NETWORK
TITLE = CALL SFC UO_MX_CIP if CIP running
//------------------------------------------------------------------------//
// SFC CALL   SFC CALL   SFC CALL   SFC CALL   SFC CALL   SFC CALL   SFC  //
//                                                                        //
// Call the SFC function if this is the running substate. This has to be  //
// called even if the block is not running so the SFC can process all     //
// commmands:                                                             //
//------------------------------------------------------------------------//
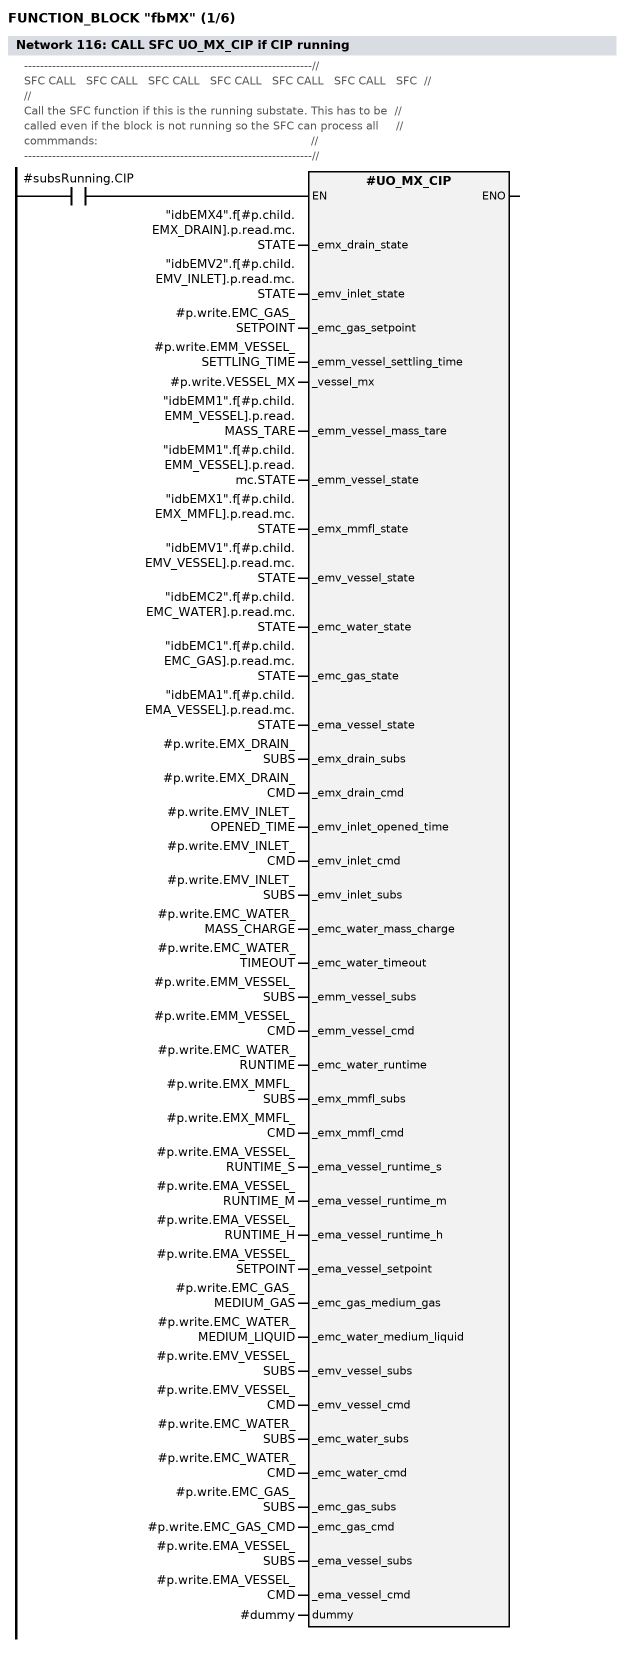
      A #subsRunning.CIP;
      JCN _notSFC_1_CIP;
      CALL #UO_MX_CIP
      (  _emx_drain_state            := "idbEMX4".f[#p.child.EMX_DRAIN].p.read.mc.STATE ,
         _emv_inlet_state            := "idbEMV2".f[#p.child.EMV_INLET].p.read.mc.STATE ,
         _emc_gas_setpoint           := #p.write.EMC_GAS_SETPOINT ,
         _emm_vessel_settling_time   := #p.write.EMM_VESSEL_SETTLING_TIME ,
         _vessel_mx                  := #p.write.VESSEL_MX ,
         _emm_vessel_mass_tare       := "idbEMM1".f[#p.child.EMM_VESSEL].p.read.MASS_TARE ,
         _emm_vessel_state           := "idbEMM1".f[#p.child.EMM_VESSEL].p.read.mc.STATE ,
         _emx_mmfl_state             := "idbEMX1".f[#p.child.EMX_MMFL].p.read.mc.STATE ,
         _emv_vessel_state           := "idbEMV1".f[#p.child.EMV_VESSEL].p.read.mc.STATE ,
         _emc_water_state            := "idbEMC2".f[#p.child.EMC_WATER].p.read.mc.STATE ,
         _emc_gas_state              := "idbEMC1".f[#p.child.EMC_GAS].p.read.mc.STATE ,
         _ema_vessel_state           := "idbEMA1".f[#p.child.EMA_VESSEL].p.read.mc.STATE ,
         _emx_drain_subs             := #p.write.EMX_DRAIN_SUBS ,
         _emx_drain_cmd              := #p.write.EMX_DRAIN_CMD ,
         _emv_inlet_opened_time      := #p.write.EMV_INLET_OPENED_TIME ,
         _emv_inlet_cmd              := #p.write.EMV_INLET_CMD ,
         _emv_inlet_subs             := #p.write.EMV_INLET_SUBS ,
         _emc_water_mass_charge      := #p.write.EMC_WATER_MASS_CHARGE ,
         _emc_water_timeout          := #p.write.EMC_WATER_TIMEOUT ,
         _emm_vessel_subs            := #p.write.EMM_VESSEL_SUBS ,
         _emm_vessel_cmd             := #p.write.EMM_VESSEL_CMD ,
         _emc_water_runtime          := #p.write.EMC_WATER_RUNTIME ,
         _emx_mmfl_subs              := #p.write.EMX_MMFL_SUBS ,
         _emx_mmfl_cmd               := #p.write.EMX_MMFL_CMD ,
         _ema_vessel_runtime_s       := #p.write.EMA_VESSEL_RUNTIME_S ,
         _ema_vessel_runtime_m       := #p.write.EMA_VESSEL_RUNTIME_M ,
         _ema_vessel_runtime_h       := #p.write.EMA_VESSEL_RUNTIME_H ,
         _ema_vessel_setpoint        := #p.write.EMA_VESSEL_SETPOINT ,
         _emc_gas_medium_gas         := #p.write.EMC_GAS_MEDIUM_GAS ,
         _emc_water_medium_liquid    := #p.write.EMC_WATER_MEDIUM_LIQUID ,
         _emv_vessel_subs            := #p.write.EMV_VESSEL_SUBS ,
         _emv_vessel_cmd             := #p.write.EMV_VESSEL_CMD ,
         _emc_water_subs             := #p.write.EMC_WATER_SUBS ,
         _emc_water_cmd              := #p.write.EMC_WATER_CMD ,
         _emc_gas_subs               := #p.write.EMC_GAS_SUBS ,
         _emc_gas_cmd                := #p.write.EMC_GAS_CMD ,
         _ema_vessel_subs            := #p.write.EMA_VESSEL_SUBS ,
         _ema_vessel_cmd             := #p.write.EMA_VESSEL_CMD ,
         dummy                       := #dummy
      );
_notSFC_1_CIP:      NOP 0;
NETWORK
TITLE = CALL SFC UO_MX_FILL if FILL running
//------------------------------------------------------------------------//
// SFC CALL   SFC CALL   SFC CALL   SFC CALL   SFC CALL   SFC CALL   SFC  //
//                                                                        //
// Call the SFC function if this is the running substate. This has to be  //
// called even if the block is not running so the SFC can process all     //
// commmands:                                                             //
//------------------------------------------------------------------------//
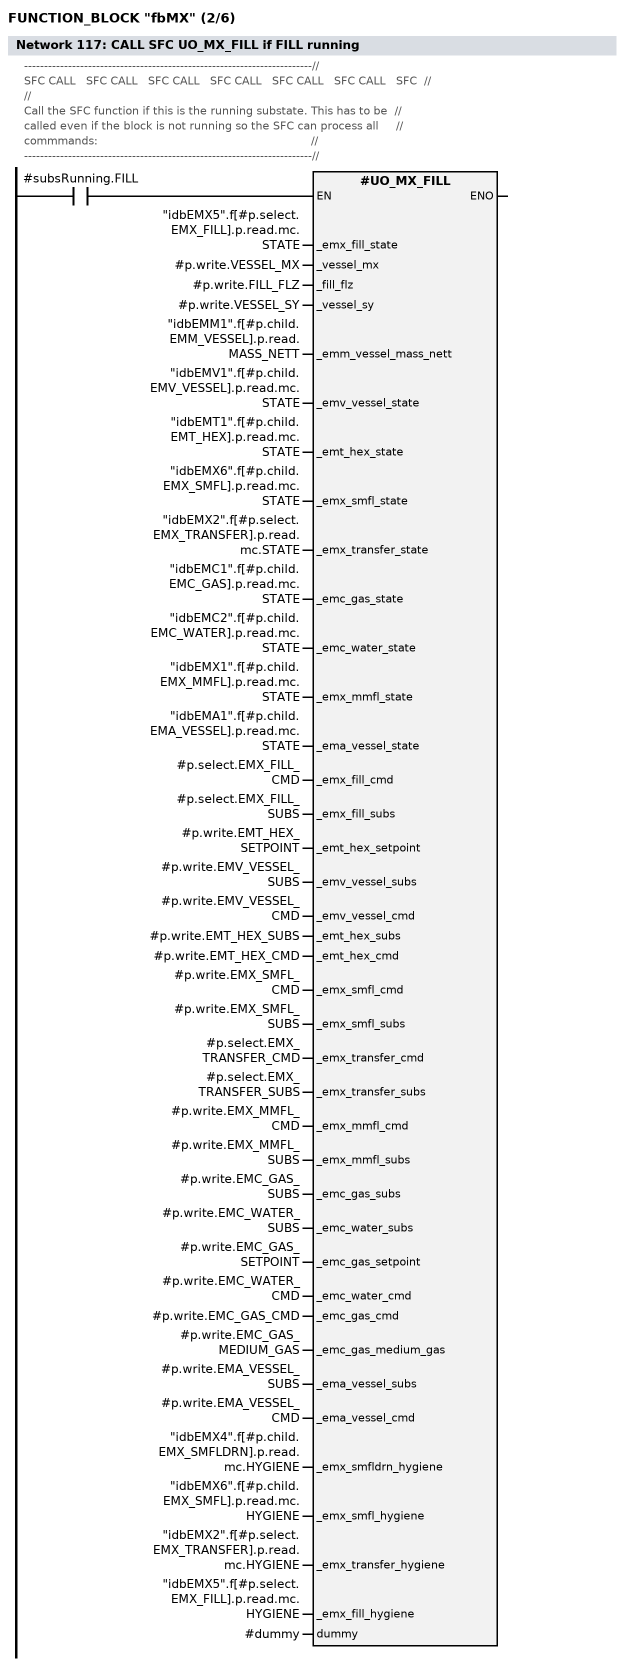
      A #subsRunning.FILL;
      JCN _notSFC_5_FILL;
      CALL #UO_MX_FILL
      (  _emx_fill_state             := "idbEMX5".f[#p.select.EMX_FILL].p.read.mc.STATE ,
         _vessel_mx                  := #p.write.VESSEL_MX ,
         _fill_flz                   := #p.write.FILL_FLZ ,
         _vessel_sy                  := #p.write.VESSEL_SY ,
         _emm_vessel_mass_nett       := "idbEMM1".f[#p.child.EMM_VESSEL].p.read.MASS_NETT ,
         _emv_vessel_state           := "idbEMV1".f[#p.child.EMV_VESSEL].p.read.mc.STATE ,
         _emt_hex_state              := "idbEMT1".f[#p.child.EMT_HEX].p.read.mc.STATE ,
         _emx_smfl_state             := "idbEMX6".f[#p.child.EMX_SMFL].p.read.mc.STATE ,
         _emx_transfer_state         := "idbEMX2".f[#p.select.EMX_TRANSFER].p.read.mc.STATE ,
         _emc_gas_state              := "idbEMC1".f[#p.child.EMC_GAS].p.read.mc.STATE ,
         _emc_water_state            := "idbEMC2".f[#p.child.EMC_WATER].p.read.mc.STATE ,
         _emx_mmfl_state             := "idbEMX1".f[#p.child.EMX_MMFL].p.read.mc.STATE ,
         _ema_vessel_state           := "idbEMA1".f[#p.child.EMA_VESSEL].p.read.mc.STATE ,
         _emx_fill_cmd               := #p.select.EMX_FILL_CMD ,
         _emx_fill_subs              := #p.select.EMX_FILL_SUBS ,
         _emt_hex_setpoint           := #p.write.EMT_HEX_SETPOINT ,
         _emv_vessel_subs            := #p.write.EMV_VESSEL_SUBS ,
         _emv_vessel_cmd             := #p.write.EMV_VESSEL_CMD ,
         _emt_hex_subs               := #p.write.EMT_HEX_SUBS ,
         _emt_hex_cmd                := #p.write.EMT_HEX_CMD ,
         _emx_smfl_cmd               := #p.write.EMX_SMFL_CMD ,
         _emx_smfl_subs              := #p.write.EMX_SMFL_SUBS ,
         _emx_transfer_cmd           := #p.select.EMX_TRANSFER_CMD ,
         _emx_transfer_subs          := #p.select.EMX_TRANSFER_SUBS ,
         _emx_mmfl_cmd               := #p.write.EMX_MMFL_CMD ,
         _emx_mmfl_subs              := #p.write.EMX_MMFL_SUBS ,
         _emc_gas_subs               := #p.write.EMC_GAS_SUBS ,
         _emc_water_subs             := #p.write.EMC_WATER_SUBS ,
         _emc_gas_setpoint           := #p.write.EMC_GAS_SETPOINT ,
         _emc_water_cmd              := #p.write.EMC_WATER_CMD ,
         _emc_gas_cmd                := #p.write.EMC_GAS_CMD ,
         _emc_gas_medium_gas         := #p.write.EMC_GAS_MEDIUM_GAS ,
         _ema_vessel_subs            := #p.write.EMA_VESSEL_SUBS ,
         _ema_vessel_cmd             := #p.write.EMA_VESSEL_CMD ,
         _emx_smfldrn_hygiene        := "idbEMX4".f[#p.child.EMX_SMFLDRN].p.read.mc.HYGIENE ,
         _emx_smfl_hygiene           := "idbEMX6".f[#p.child.EMX_SMFL].p.read.mc.HYGIENE ,
         _emx_transfer_hygiene       := "idbEMX2".f[#p.select.EMX_TRANSFER].p.read.mc.HYGIENE ,
         _emx_fill_hygiene           := "idbEMX5".f[#p.select.EMX_FILL].p.read.mc.HYGIENE ,
         dummy                       := #dummy
      );
_notSFC_5_FILL:      NOP 0;
NETWORK
TITLE = CALL SFC UO_MX_FILTER if FILTER running
//------------------------------------------------------------------------//
// SFC CALL   SFC CALL   SFC CALL   SFC CALL   SFC CALL   SFC CALL   SFC  //
//                                                                        //
// Call the SFC function if this is the running substate. This has to be  //
// called even if the block is not running so the SFC can process all     //
// commmands:                                                             //
//------------------------------------------------------------------------//
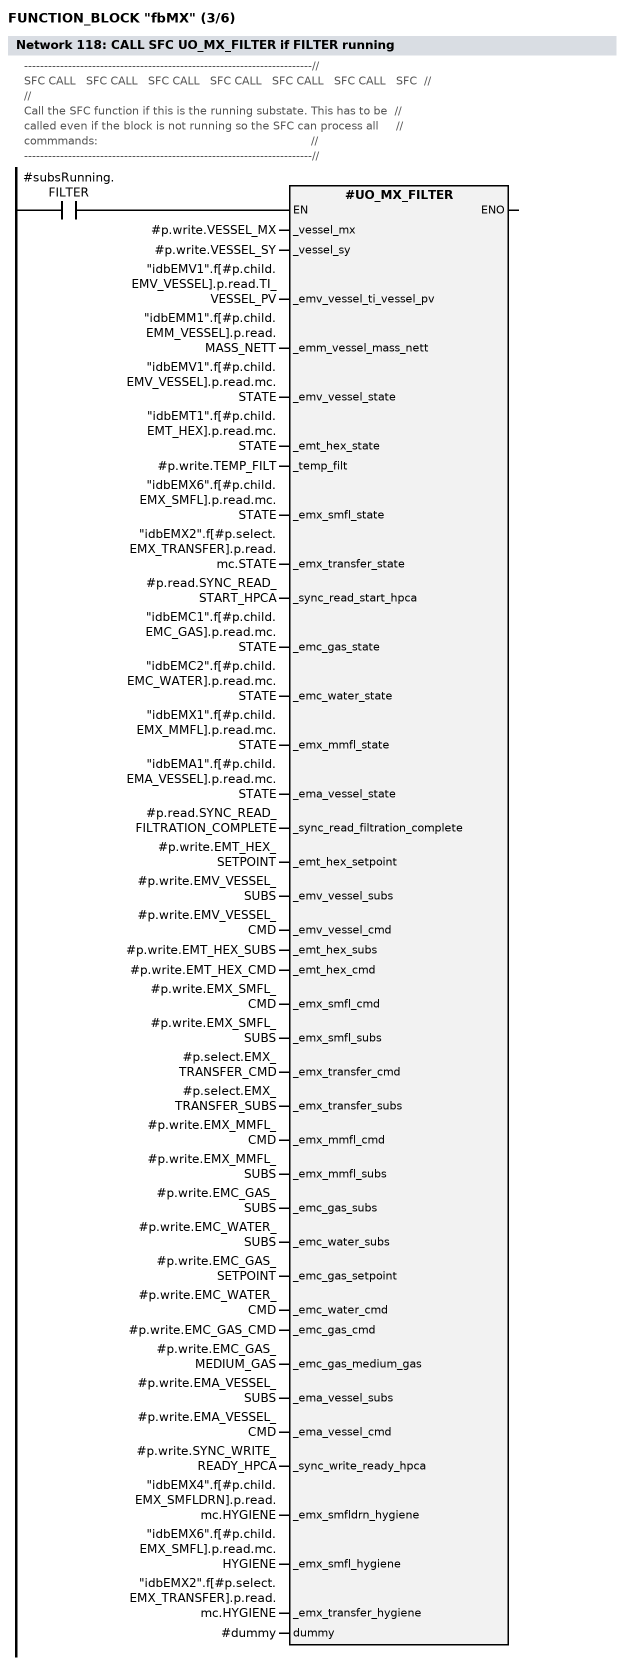
      A #subsRunning.FILTER;
      JCN _notSFC_3_FILTER;
      CALL #UO_MX_FILTER
      (  _vessel_mx                  := #p.write.VESSEL_MX ,
         _vessel_sy                  := #p.write.VESSEL_SY ,
         _emv_vessel_ti_vessel_pv    := "idbEMV1".f[#p.child.EMV_VESSEL].p.read.TI_VESSEL_PV ,
         _emm_vessel_mass_nett       := "idbEMM1".f[#p.child.EMM_VESSEL].p.read.MASS_NETT ,
         _emv_vessel_state           := "idbEMV1".f[#p.child.EMV_VESSEL].p.read.mc.STATE ,
         _emt_hex_state              := "idbEMT1".f[#p.child.EMT_HEX].p.read.mc.STATE ,
         _temp_filt                  := #p.write.TEMP_FILT ,
         _emx_smfl_state             := "idbEMX6".f[#p.child.EMX_SMFL].p.read.mc.STATE ,
         _emx_transfer_state         := "idbEMX2".f[#p.select.EMX_TRANSFER].p.read.mc.STATE ,
         _sync_read_start_hpca       := #p.read.SYNC_READ_START_HPCA ,
         _emc_gas_state              := "idbEMC1".f[#p.child.EMC_GAS].p.read.mc.STATE ,
         _emc_water_state            := "idbEMC2".f[#p.child.EMC_WATER].p.read.mc.STATE ,
         _emx_mmfl_state             := "idbEMX1".f[#p.child.EMX_MMFL].p.read.mc.STATE ,
         _ema_vessel_state           := "idbEMA1".f[#p.child.EMA_VESSEL].p.read.mc.STATE ,
         _sync_read_filtration_complete:= #p.read.SYNC_READ_FILTRATION_COMPLETE ,
         _emt_hex_setpoint           := #p.write.EMT_HEX_SETPOINT ,
         _emv_vessel_subs            := #p.write.EMV_VESSEL_SUBS ,
         _emv_vessel_cmd             := #p.write.EMV_VESSEL_CMD ,
         _emt_hex_subs               := #p.write.EMT_HEX_SUBS ,
         _emt_hex_cmd                := #p.write.EMT_HEX_CMD ,
         _emx_smfl_cmd               := #p.write.EMX_SMFL_CMD ,
         _emx_smfl_subs              := #p.write.EMX_SMFL_SUBS ,
         _emx_transfer_cmd           := #p.select.EMX_TRANSFER_CMD ,
         _emx_transfer_subs          := #p.select.EMX_TRANSFER_SUBS ,
         _emx_mmfl_cmd               := #p.write.EMX_MMFL_CMD ,
         _emx_mmfl_subs              := #p.write.EMX_MMFL_SUBS ,
         _emc_gas_subs               := #p.write.EMC_GAS_SUBS ,
         _emc_water_subs             := #p.write.EMC_WATER_SUBS ,
         _emc_gas_setpoint           := #p.write.EMC_GAS_SETPOINT ,
         _emc_water_cmd              := #p.write.EMC_WATER_CMD ,
         _emc_gas_cmd                := #p.write.EMC_GAS_CMD ,
         _emc_gas_medium_gas         := #p.write.EMC_GAS_MEDIUM_GAS ,
         _ema_vessel_subs            := #p.write.EMA_VESSEL_SUBS ,
         _ema_vessel_cmd             := #p.write.EMA_VESSEL_CMD ,
         _sync_write_ready_hpca      := #p.write.SYNC_WRITE_READY_HPCA ,
         _emx_smfldrn_hygiene        := "idbEMX4".f[#p.child.EMX_SMFLDRN].p.read.mc.HYGIENE ,
         _emx_smfl_hygiene           := "idbEMX6".f[#p.child.EMX_SMFL].p.read.mc.HYGIENE ,
         _emx_transfer_hygiene       := "idbEMX2".f[#p.select.EMX_TRANSFER].p.read.mc.HYGIENE ,
         dummy                       := #dummy
      );
_notSFC_3_FILTER:      NOP 0;
NETWORK
TITLE = CALL SFC UO_MX_MAKE if MAKE running
//------------------------------------------------------------------------//
// SFC CALL   SFC CALL   SFC CALL   SFC CALL   SFC CALL   SFC CALL   SFC  //
//                                                                        //
// Call the SFC function if this is the running substate. This has to be  //
// called even if the block is not running so the SFC can process all     //
// commmands:                                                             //
//------------------------------------------------------------------------//
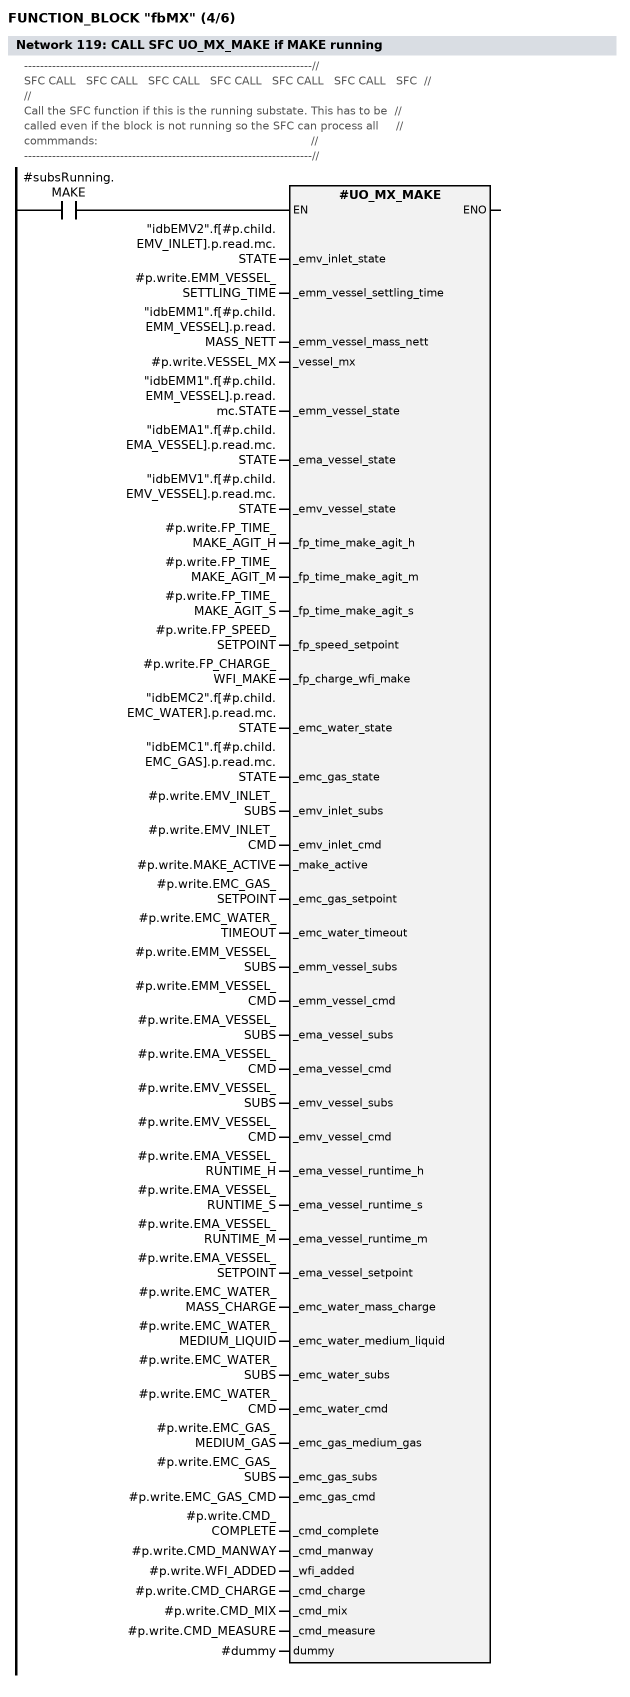
      A #subsRunning.MAKE;
      JCN _notSFC_1_MAKE;
      CALL #UO_MX_MAKE
      (  _emv_inlet_state            := "idbEMV2".f[#p.child.EMV_INLET].p.read.mc.STATE ,
         _emm_vessel_settling_time   := #p.write.EMM_VESSEL_SETTLING_TIME ,
         _emm_vessel_mass_nett       := "idbEMM1".f[#p.child.EMM_VESSEL].p.read.MASS_NETT ,
         _vessel_mx                  := #p.write.VESSEL_MX ,
         _emm_vessel_state           := "idbEMM1".f[#p.child.EMM_VESSEL].p.read.mc.STATE ,
         _ema_vessel_state           := "idbEMA1".f[#p.child.EMA_VESSEL].p.read.mc.STATE ,
         _emv_vessel_state           := "idbEMV1".f[#p.child.EMV_VESSEL].p.read.mc.STATE ,
         _fp_time_make_agit_h        := #p.write.FP_TIME_MAKE_AGIT_H ,
         _fp_time_make_agit_m        := #p.write.FP_TIME_MAKE_AGIT_M ,
         _fp_time_make_agit_s        := #p.write.FP_TIME_MAKE_AGIT_S ,
         _fp_speed_setpoint          := #p.write.FP_SPEED_SETPOINT ,
         _fp_charge_wfi_make         := #p.write.FP_CHARGE_WFI_MAKE ,
         _emc_water_state            := "idbEMC2".f[#p.child.EMC_WATER].p.read.mc.STATE ,
         _emc_gas_state              := "idbEMC1".f[#p.child.EMC_GAS].p.read.mc.STATE ,
         _emv_inlet_subs             := #p.write.EMV_INLET_SUBS ,
         _emv_inlet_cmd              := #p.write.EMV_INLET_CMD ,
         _make_active                := #p.write.MAKE_ACTIVE ,
         _emc_gas_setpoint           := #p.write.EMC_GAS_SETPOINT ,
         _emc_water_timeout          := #p.write.EMC_WATER_TIMEOUT ,
         _emm_vessel_subs            := #p.write.EMM_VESSEL_SUBS ,
         _emm_vessel_cmd             := #p.write.EMM_VESSEL_CMD ,
         _ema_vessel_subs            := #p.write.EMA_VESSEL_SUBS ,
         _ema_vessel_cmd             := #p.write.EMA_VESSEL_CMD ,
         _emv_vessel_subs            := #p.write.EMV_VESSEL_SUBS ,
         _emv_vessel_cmd             := #p.write.EMV_VESSEL_CMD ,
         _ema_vessel_runtime_h       := #p.write.EMA_VESSEL_RUNTIME_H ,
         _ema_vessel_runtime_s       := #p.write.EMA_VESSEL_RUNTIME_S ,
         _ema_vessel_runtime_m       := #p.write.EMA_VESSEL_RUNTIME_M ,
         _ema_vessel_setpoint        := #p.write.EMA_VESSEL_SETPOINT ,
         _emc_water_mass_charge      := #p.write.EMC_WATER_MASS_CHARGE ,
         _emc_water_medium_liquid    := #p.write.EMC_WATER_MEDIUM_LIQUID ,
         _emc_water_subs             := #p.write.EMC_WATER_SUBS ,
         _emc_water_cmd              := #p.write.EMC_WATER_CMD ,
         _emc_gas_medium_gas         := #p.write.EMC_GAS_MEDIUM_GAS ,
         _emc_gas_subs               := #p.write.EMC_GAS_SUBS ,
         _emc_gas_cmd                := #p.write.EMC_GAS_CMD ,
         _cmd_complete               := #p.write.CMD_COMPLETE ,
         _cmd_manway                 := #p.write.CMD_MANWAY ,
         _wfi_added                  := #p.write.WFI_ADDED ,
         _cmd_charge                 := #p.write.CMD_CHARGE ,
         _cmd_mix                    := #p.write.CMD_MIX ,
         _cmd_measure                := #p.write.CMD_MEASURE ,
         dummy                       := #dummy
      );
_notSFC_1_MAKE:      NOP 0;
NETWORK
TITLE = CALL SFC UO_MX_SETUP if SETUP running
//------------------------------------------------------------------------//
// SFC CALL   SFC CALL   SFC CALL   SFC CALL   SFC CALL   SFC CALL   SFC  //
//                                                                        //
// Call the SFC function if this is the running substate. This has to be  //
// called even if the block is not running so the SFC can process all     //
// commmands:                                                             //
//------------------------------------------------------------------------//
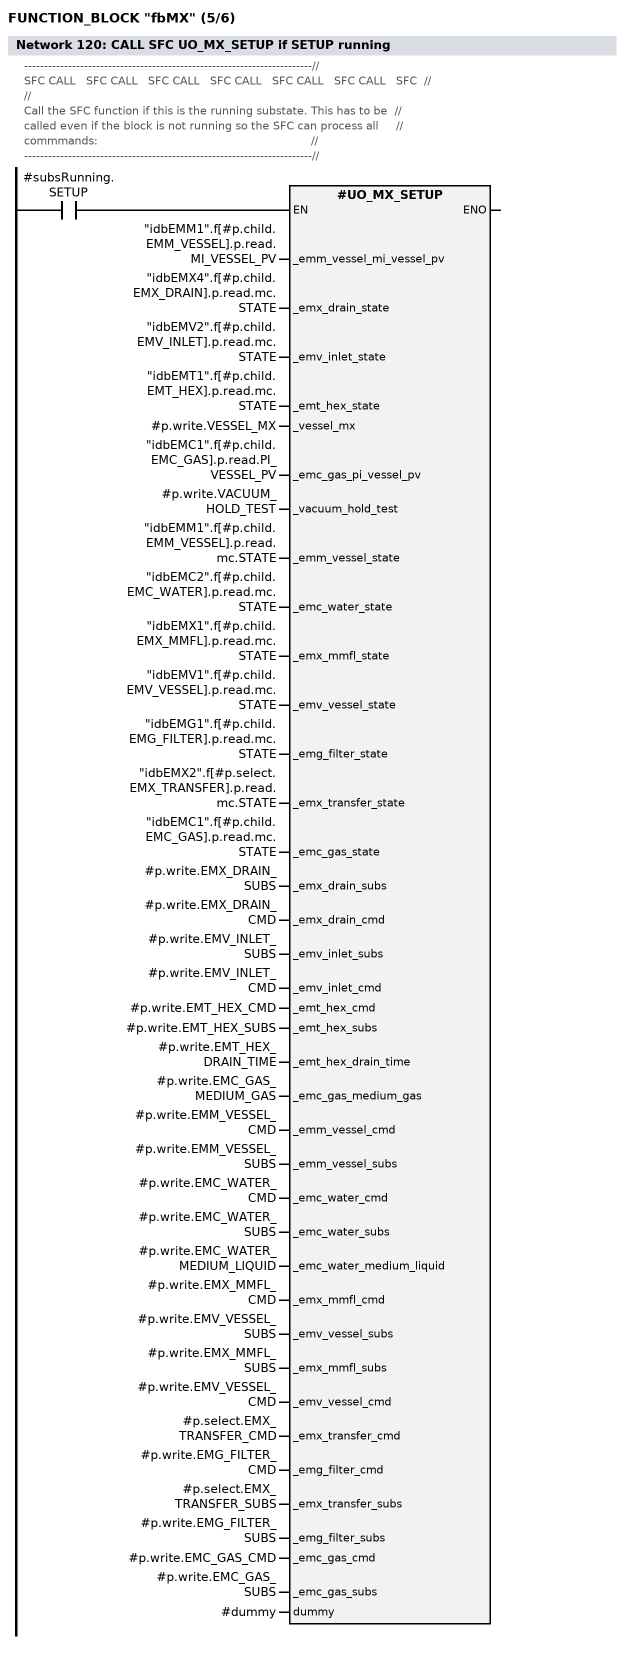
      A #subsRunning.SETUP;
      JCN _notSFC_3_SETUP;
      CALL #UO_MX_SETUP
      (  _emm_vessel_mi_vessel_pv    := "idbEMM1".f[#p.child.EMM_VESSEL].p.read.MI_VESSEL_PV ,
         _emx_drain_state            := "idbEMX4".f[#p.child.EMX_DRAIN].p.read.mc.STATE ,
         _emv_inlet_state            := "idbEMV2".f[#p.child.EMV_INLET].p.read.mc.STATE ,
         _emt_hex_state              := "idbEMT1".f[#p.child.EMT_HEX].p.read.mc.STATE ,
         _vessel_mx                  := #p.write.VESSEL_MX ,
         _emc_gas_pi_vessel_pv       := "idbEMC1".f[#p.child.EMC_GAS].p.read.PI_VESSEL_PV ,
         _vacuum_hold_test           := #p.write.VACUUM_HOLD_TEST ,
         _emm_vessel_state           := "idbEMM1".f[#p.child.EMM_VESSEL].p.read.mc.STATE ,
         _emc_water_state            := "idbEMC2".f[#p.child.EMC_WATER].p.read.mc.STATE ,
         _emx_mmfl_state             := "idbEMX1".f[#p.child.EMX_MMFL].p.read.mc.STATE ,
         _emv_vessel_state           := "idbEMV1".f[#p.child.EMV_VESSEL].p.read.mc.STATE ,
         _emg_filter_state           := "idbEMG1".f[#p.child.EMG_FILTER].p.read.mc.STATE ,
         _emx_transfer_state         := "idbEMX2".f[#p.select.EMX_TRANSFER].p.read.mc.STATE ,
         _emc_gas_state              := "idbEMC1".f[#p.child.EMC_GAS].p.read.mc.STATE ,
         _emx_drain_subs             := #p.write.EMX_DRAIN_SUBS ,
         _emx_drain_cmd              := #p.write.EMX_DRAIN_CMD ,
         _emv_inlet_subs             := #p.write.EMV_INLET_SUBS ,
         _emv_inlet_cmd              := #p.write.EMV_INLET_CMD ,
         _emt_hex_cmd                := #p.write.EMT_HEX_CMD ,
         _emt_hex_subs               := #p.write.EMT_HEX_SUBS ,
         _emt_hex_drain_time         := #p.write.EMT_HEX_DRAIN_TIME ,
         _emc_gas_medium_gas         := #p.write.EMC_GAS_MEDIUM_GAS ,
         _emm_vessel_cmd             := #p.write.EMM_VESSEL_CMD ,
         _emm_vessel_subs            := #p.write.EMM_VESSEL_SUBS ,
         _emc_water_cmd              := #p.write.EMC_WATER_CMD ,
         _emc_water_subs             := #p.write.EMC_WATER_SUBS ,
         _emc_water_medium_liquid    := #p.write.EMC_WATER_MEDIUM_LIQUID ,
         _emx_mmfl_cmd               := #p.write.EMX_MMFL_CMD ,
         _emv_vessel_subs            := #p.write.EMV_VESSEL_SUBS ,
         _emx_mmfl_subs              := #p.write.EMX_MMFL_SUBS ,
         _emv_vessel_cmd             := #p.write.EMV_VESSEL_CMD ,
         _emx_transfer_cmd           := #p.select.EMX_TRANSFER_CMD ,
         _emg_filter_cmd             := #p.write.EMG_FILTER_CMD ,
         _emx_transfer_subs          := #p.select.EMX_TRANSFER_SUBS ,
         _emg_filter_subs            := #p.write.EMG_FILTER_SUBS ,
         _emc_gas_cmd                := #p.write.EMC_GAS_CMD ,
         _emc_gas_subs               := #p.write.EMC_GAS_SUBS ,
         dummy                       := #dummy
      );
_notSFC_3_SETUP:      NOP 0;
NETWORK
TITLE = CALL SFC UO_MX_SIP if SIP running
//------------------------------------------------------------------------//
// SFC CALL   SFC CALL   SFC CALL   SFC CALL   SFC CALL   SFC CALL   SFC  //
//                                                                        //
// Call the SFC function if this is the running substate. This has to be  //
// called even if the block is not running so the SFC can process all     //
// commmands:                                                             //
//------------------------------------------------------------------------//
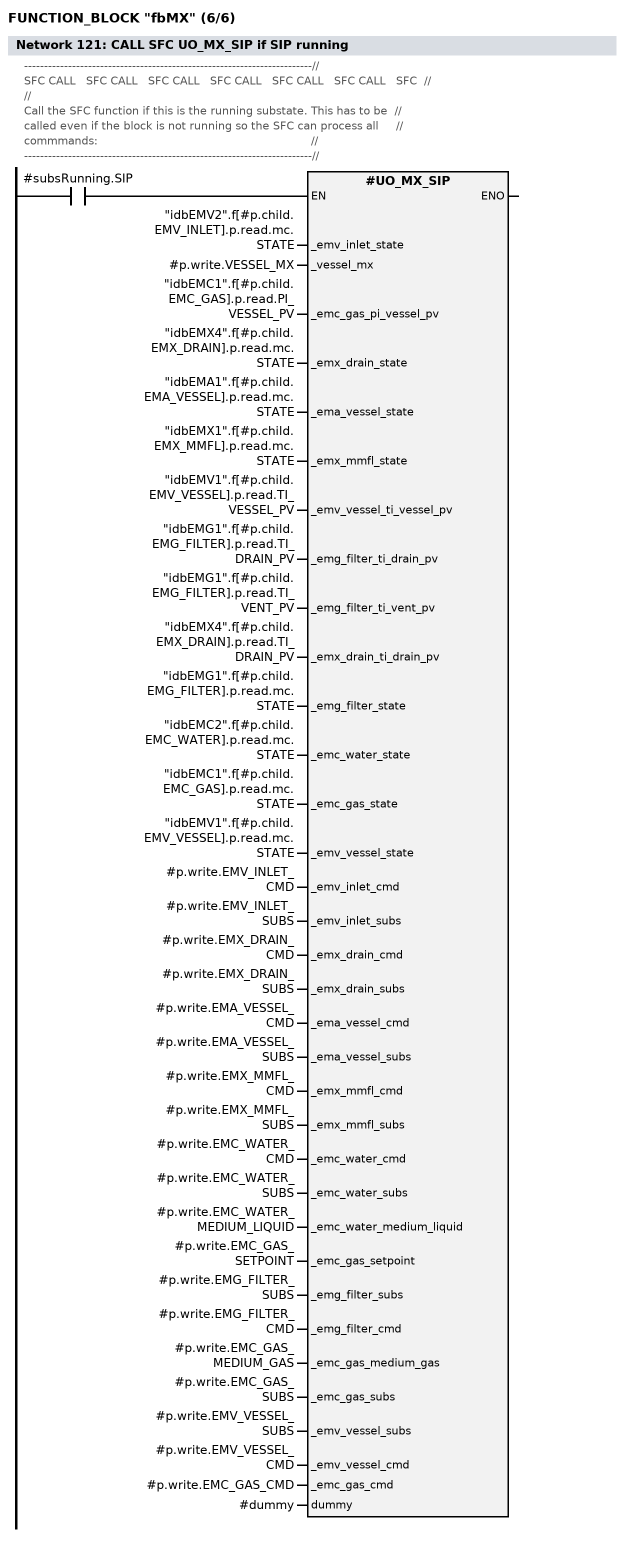
      A #subsRunning.SIP;
      JCN _notSFC_1_SIP;
      CALL #UO_MX_SIP
      (  _emv_inlet_state            := "idbEMV2".f[#p.child.EMV_INLET].p.read.mc.STATE ,
         _vessel_mx                  := #p.write.VESSEL_MX ,
         _emc_gas_pi_vessel_pv       := "idbEMC1".f[#p.child.EMC_GAS].p.read.PI_VESSEL_PV ,
         _emx_drain_state            := "idbEMX4".f[#p.child.EMX_DRAIN].p.read.mc.STATE ,
         _ema_vessel_state           := "idbEMA1".f[#p.child.EMA_VESSEL].p.read.mc.STATE ,
         _emx_mmfl_state             := "idbEMX1".f[#p.child.EMX_MMFL].p.read.mc.STATE ,
         _emv_vessel_ti_vessel_pv    := "idbEMV1".f[#p.child.EMV_VESSEL].p.read.TI_VESSEL_PV ,
         _emg_filter_ti_drain_pv     := "idbEMG1".f[#p.child.EMG_FILTER].p.read.TI_DRAIN_PV ,
         _emg_filter_ti_vent_pv      := "idbEMG1".f[#p.child.EMG_FILTER].p.read.TI_VENT_PV ,
         _emx_drain_ti_drain_pv      := "idbEMX4".f[#p.child.EMX_DRAIN].p.read.TI_DRAIN_PV ,
         _emg_filter_state           := "idbEMG1".f[#p.child.EMG_FILTER].p.read.mc.STATE ,
         _emc_water_state            := "idbEMC2".f[#p.child.EMC_WATER].p.read.mc.STATE ,
         _emc_gas_state              := "idbEMC1".f[#p.child.EMC_GAS].p.read.mc.STATE ,
         _emv_vessel_state           := "idbEMV1".f[#p.child.EMV_VESSEL].p.read.mc.STATE ,
         _emv_inlet_cmd              := #p.write.EMV_INLET_CMD ,
         _emv_inlet_subs             := #p.write.EMV_INLET_SUBS ,
         _emx_drain_cmd              := #p.write.EMX_DRAIN_CMD ,
         _emx_drain_subs             := #p.write.EMX_DRAIN_SUBS ,
         _ema_vessel_cmd             := #p.write.EMA_VESSEL_CMD ,
         _ema_vessel_subs            := #p.write.EMA_VESSEL_SUBS ,
         _emx_mmfl_cmd               := #p.write.EMX_MMFL_CMD ,
         _emx_mmfl_subs              := #p.write.EMX_MMFL_SUBS ,
         _emc_water_cmd              := #p.write.EMC_WATER_CMD ,
         _emc_water_subs             := #p.write.EMC_WATER_SUBS ,
         _emc_water_medium_liquid    := #p.write.EMC_WATER_MEDIUM_LIQUID ,
         _emc_gas_setpoint           := #p.write.EMC_GAS_SETPOINT ,
         _emg_filter_subs            := #p.write.EMG_FILTER_SUBS ,
         _emg_filter_cmd             := #p.write.EMG_FILTER_CMD ,
         _emc_gas_medium_gas         := #p.write.EMC_GAS_MEDIUM_GAS ,
         _emc_gas_subs               := #p.write.EMC_GAS_SUBS ,
         _emv_vessel_subs            := #p.write.EMV_VESSEL_SUBS ,
         _emv_vessel_cmd             := #p.write.EMV_VESSEL_CMD ,
         _emc_gas_cmd                := #p.write.EMC_GAS_CMD ,
         dummy                       := #dummy
      );
_notSFC_1_SIP:      NOP 0;

NETWORK
TITLE = Check if any Child state does not match the command
//------------------------------------------------------------------------//
// CHILD FLOWPATH STATE MISMATCH   CHILD FLOWPATH STATE MISMATCH   CHILD  //
//                                                                        //
// Check if any child flowpath device state does not match the command    //
// from this parent block if the child state grace period timer has       //
// expired. Stop checking if the first child state mismatch found:        //
//------------------------------------------------------------------------//
      A(;
      O(;
      A "alwaysHigh";
      A "idbEMA1".f[#p.child.EMA_VESSEL].p.write.mc.ARMED;
      A "idbEMA1".f[#p.child.EMA_VESSEL].p.read.mc.FLOWPATH;
      A(;
      L "idbEMA1".f[#p.child.EMA_VESSEL].p.read.mc.STATE;
      L #childReqCMD.EMA_VESSEL;
      <>I;
      );
      A(;
      L "idbEMA1".f[#p.child.EMA_VESSEL].p.read.mc.STATE;
      L "dbCONST".BLK.STATE.COMPLETED;
      <>I;
      );
      AN(;
      A(;
      L "dbCONST".BLK.CMD.START;
      L #childReqCMD.EMA_VESSEL;
      ==I;
      );
      A(;
      L "idbEMA1".f[#p.child.EMA_VESSEL].p.read.mc.STATE;
      L "idbEMA1".f[#p.child.EMA_VESSEL].p.write.mc.SUBS;
      ==I;
      );
      );
      );
      O(;
      A "alwaysHigh";
      A "idbEMC1".f[#p.child.EMC_GAS].p.write.mc.ARMED;
      A "idbEMC1".f[#p.child.EMC_GAS].p.read.mc.FLOWPATH;
      A(;
      L "idbEMC1".f[#p.child.EMC_GAS].p.read.mc.STATE;
      L #childReqCMD.EMC_GAS;
      <>I;
      );
      A(;
      L "idbEMC1".f[#p.child.EMC_GAS].p.read.mc.STATE;
      L "dbCONST".BLK.STATE.COMPLETED;
      <>I;
      );
      AN(;
      A(;
      L "dbCONST".BLK.CMD.START;
      L #childReqCMD.EMC_GAS;
      ==I;
      );
      A(;
      L "idbEMC1".f[#p.child.EMC_GAS].p.read.mc.STATE;
      L "idbEMC1".f[#p.child.EMC_GAS].p.write.mc.SUBS;
      ==I;
      );
      );
      );
      O(;
      A "alwaysHigh";
      A "idbEMC2".f[#p.child.EMC_WATER].p.write.mc.ARMED;
      A "idbEMC2".f[#p.child.EMC_WATER].p.read.mc.FLOWPATH;
      A(;
      L "idbEMC2".f[#p.child.EMC_WATER].p.read.mc.STATE;
      L #childReqCMD.EMC_WATER;
      <>I;
      );
      A(;
      L "idbEMC2".f[#p.child.EMC_WATER].p.read.mc.STATE;
      L "dbCONST".BLK.STATE.COMPLETED;
      <>I;
      );
      AN(;
      A(;
      L "dbCONST".BLK.CMD.START;
      L #childReqCMD.EMC_WATER;
      ==I;
      );
      A(;
      L "idbEMC2".f[#p.child.EMC_WATER].p.read.mc.STATE;
      L "idbEMC2".f[#p.child.EMC_WATER].p.write.mc.SUBS;
      ==I;
      );
      );
      );
      O(;
      A "alwaysHigh";
      A "idbEMG1".f[#p.child.EMG_FILTER].p.write.mc.ARMED;
      A "idbEMG1".f[#p.child.EMG_FILTER].p.read.mc.FLOWPATH;
      A(;
      L "idbEMG1".f[#p.child.EMG_FILTER].p.read.mc.STATE;
      L #childReqCMD.EMG_FILTER;
      <>I;
      );
      A(;
      L "idbEMG1".f[#p.child.EMG_FILTER].p.read.mc.STATE;
      L "dbCONST".BLK.STATE.COMPLETED;
      <>I;
      );
      AN(;
      A(;
      L "dbCONST".BLK.CMD.START;
      L #childReqCMD.EMG_FILTER;
      ==I;
      );
      A(;
      L "idbEMG1".f[#p.child.EMG_FILTER].p.read.mc.STATE;
      L "idbEMG1".f[#p.child.EMG_FILTER].p.write.mc.SUBS;
      ==I;
      );
      );
      );
      O(;
      A "alwaysHigh";
      A "idbEMM1".f[#p.child.EMM_VESSEL].p.write.mc.ARMED;
      A "idbEMM1".f[#p.child.EMM_VESSEL].p.read.mc.FLOWPATH;
      A(;
      L "idbEMM1".f[#p.child.EMM_VESSEL].p.read.mc.STATE;
      L #childReqCMD.EMM_VESSEL;
      <>I;
      );
      A(;
      L "idbEMM1".f[#p.child.EMM_VESSEL].p.read.mc.STATE;
      L "dbCONST".BLK.STATE.COMPLETED;
      <>I;
      );
      AN(;
      A(;
      L "dbCONST".BLK.CMD.START;
      L #childReqCMD.EMM_VESSEL;
      ==I;
      );
      A(;
      L "idbEMM1".f[#p.child.EMM_VESSEL].p.read.mc.STATE;
      L "idbEMM1".f[#p.child.EMM_VESSEL].p.write.mc.SUBS;
      ==I;
      );
      );
      );
      O(;
      A "alwaysHigh";
      A "idbEMT1".f[#p.child.EMT_HEX].p.write.mc.ARMED;
      A "idbEMT1".f[#p.child.EMT_HEX].p.read.mc.FLOWPATH;
      A(;
      L "idbEMT1".f[#p.child.EMT_HEX].p.read.mc.STATE;
      L #childReqCMD.EMT_HEX;
      <>I;
      );
      A(;
      L "idbEMT1".f[#p.child.EMT_HEX].p.read.mc.STATE;
      L "dbCONST".BLK.STATE.COMPLETED;
      <>I;
      );
      AN(;
      A(;
      L "dbCONST".BLK.CMD.START;
      L #childReqCMD.EMT_HEX;
      ==I;
      );
      A(;
      L "idbEMT1".f[#p.child.EMT_HEX].p.read.mc.STATE;
      L "idbEMT1".f[#p.child.EMT_HEX].p.write.mc.SUBS;
      ==I;
      );
      );
      );
      O(;
      A "alwaysHigh";
      A "idbEMV2".f[#p.child.EMV_INLET].p.write.mc.ARMED;
      A "idbEMV2".f[#p.child.EMV_INLET].p.read.mc.FLOWPATH;
      A(;
      L "idbEMV2".f[#p.child.EMV_INLET].p.read.mc.STATE;
      L #childReqCMD.EMV_INLET;
      <>I;
      );
      A(;
      L "idbEMV2".f[#p.child.EMV_INLET].p.read.mc.STATE;
      L "dbCONST".BLK.STATE.COMPLETED;
      <>I;
      );
      AN(;
      A(;
      L "dbCONST".BLK.CMD.START;
      L #childReqCMD.EMV_INLET;
      ==I;
      );
      A(;
      L "idbEMV2".f[#p.child.EMV_INLET].p.read.mc.STATE;
      L "idbEMV2".f[#p.child.EMV_INLET].p.write.mc.SUBS;
      ==I;
      );
      );
      );
      O(;
      A "alwaysHigh";
      A "idbEMV1".f[#p.child.EMV_VESSEL].p.write.mc.ARMED;
      A "idbEMV1".f[#p.child.EMV_VESSEL].p.read.mc.FLOWPATH;
      A(;
      L "idbEMV1".f[#p.child.EMV_VESSEL].p.read.mc.STATE;
      L #childReqCMD.EMV_VESSEL;
      <>I;
      );
      A(;
      L "idbEMV1".f[#p.child.EMV_VESSEL].p.read.mc.STATE;
      L "dbCONST".BLK.STATE.COMPLETED;
      <>I;
      );
      AN(;
      A(;
      L "dbCONST".BLK.CMD.START;
      L #childReqCMD.EMV_VESSEL;
      ==I;
      );
      A(;
      L "idbEMV1".f[#p.child.EMV_VESSEL].p.read.mc.STATE;
      L "idbEMV1".f[#p.child.EMV_VESSEL].p.write.mc.SUBS;
      ==I;
      );
      );
      );
      O(;
      A "alwaysHigh";
      A "idbEMX4".f[#p.child.EMX_DRAIN].p.write.mc.ARMED;
      A "idbEMX4".f[#p.child.EMX_DRAIN].p.read.mc.FLOWPATH;
      A(;
      L "idbEMX4".f[#p.child.EMX_DRAIN].p.read.mc.STATE;
      L #childReqCMD.EMX_DRAIN;
      <>I;
      );
      A(;
      L "idbEMX4".f[#p.child.EMX_DRAIN].p.read.mc.STATE;
      L "dbCONST".BLK.STATE.COMPLETED;
      <>I;
      );
      AN(;
      A(;
      L "dbCONST".BLK.CMD.START;
      L #childReqCMD.EMX_DRAIN;
      ==I;
      );
      A(;
      L "idbEMX4".f[#p.child.EMX_DRAIN].p.read.mc.STATE;
      L "idbEMX4".f[#p.child.EMX_DRAIN].p.write.mc.SUBS;
      ==I;
      );
      );
      );
      O(;
      A #selected_FILL_FLZ.FL1;
      A "idbEMX5".f[#p.child.EMX_FILL1].p.write.mc.ARMED;
      A "idbEMX5".f[#p.child.EMX_FILL1].p.read.mc.FLOWPATH;
      A(;
      L "idbEMX5".f[#p.child.EMX_FILL1].p.read.mc.STATE;
      L #childReqCMD.EMX_FILL1;
      <>I;
      );
      A(;
      L "idbEMX5".f[#p.child.EMX_FILL1].p.read.mc.STATE;
      L "dbCONST".BLK.STATE.COMPLETED;
      <>I;
      );
      AN(;
      A(;
      L "dbCONST".BLK.CMD.START;
      L #childReqCMD.EMX_FILL1;
      ==I;
      );
      A(;
      L "idbEMX5".f[#p.child.EMX_FILL1].p.read.mc.STATE;
      L "idbEMX5".f[#p.child.EMX_FILL1].p.write.mc.SUBS;
      ==I;
      );
      );
      );
      O(;
      A #selected_FILL_FLZ.FL2;
      A "idbEMX5".f[#p.child.EMX_FILL2].p.write.mc.ARMED;
      A "idbEMX5".f[#p.child.EMX_FILL2].p.read.mc.FLOWPATH;
      A(;
      L "idbEMX5".f[#p.child.EMX_FILL2].p.read.mc.STATE;
      L #childReqCMD.EMX_FILL2;
      <>I;
      );
      A(;
      L "idbEMX5".f[#p.child.EMX_FILL2].p.read.mc.STATE;
      L "dbCONST".BLK.STATE.COMPLETED;
      <>I;
      );
      AN(;
      A(;
      L "dbCONST".BLK.CMD.START;
      L #childReqCMD.EMX_FILL2;
      ==I;
      );
      A(;
      L "idbEMX5".f[#p.child.EMX_FILL2].p.read.mc.STATE;
      L "idbEMX5".f[#p.child.EMX_FILL2].p.write.mc.SUBS;
      ==I;
      );
      );
      );
      O(;
      A "alwaysHigh";
      A "idbEMX1".f[#p.child.EMX_MMFL].p.write.mc.ARMED;
      A "idbEMX1".f[#p.child.EMX_MMFL].p.read.mc.FLOWPATH;
      A(;
      L "idbEMX1".f[#p.child.EMX_MMFL].p.read.mc.STATE;
      L #childReqCMD.EMX_MMFL;
      <>I;
      );
      A(;
      L "idbEMX1".f[#p.child.EMX_MMFL].p.read.mc.STATE;
      L "dbCONST".BLK.STATE.COMPLETED;
      <>I;
      );
      AN(;
      A(;
      L "dbCONST".BLK.CMD.START;
      L #childReqCMD.EMX_MMFL;
      ==I;
      );
      A(;
      L "idbEMX1".f[#p.child.EMX_MMFL].p.read.mc.STATE;
      L "idbEMX1".f[#p.child.EMX_MMFL].p.write.mc.SUBS;
      ==I;
      );
      );
      );
      O(;
      O #selected_FILL_FLZ.FL1;
      O #selected_FILL_FLZ.FL2;
      O #selected_VESSEL_SY.S1;
      O #selected_VESSEL_SY.S2;
      A "idbEMX6".f[#p.child.EMX_SMFL].p.write.mc.ARMED;
      A "idbEMX6".f[#p.child.EMX_SMFL].p.read.mc.FLOWPATH;
      A(;
      L "idbEMX6".f[#p.child.EMX_SMFL].p.read.mc.STATE;
      L #childReqCMD.EMX_SMFL;
      <>I;
      );
      A(;
      L "idbEMX6".f[#p.child.EMX_SMFL].p.read.mc.STATE;
      L "dbCONST".BLK.STATE.COMPLETED;
      <>I;
      );
      AN(;
      A(;
      L "dbCONST".BLK.CMD.START;
      L #childReqCMD.EMX_SMFL;
      ==I;
      );
      A(;
      L "idbEMX6".f[#p.child.EMX_SMFL].p.read.mc.STATE;
      L "idbEMX6".f[#p.child.EMX_SMFL].p.write.mc.SUBS;
      ==I;
      );
      );
      );
      O(;
      O #selected_FILL_FLZ.FL1;
      O #selected_FILL_FLZ.FL2;
      O #selected_VESSEL_SY.S1;
      O #selected_VESSEL_SY.S2;
      A "idbEMX4".f[#p.child.EMX_SMFLDRN].p.write.mc.ARMED;
      A "idbEMX4".f[#p.child.EMX_SMFLDRN].p.read.mc.FLOWPATH;
      A(;
      L "idbEMX4".f[#p.child.EMX_SMFLDRN].p.read.mc.STATE;
      L #childReqCMD.EMX_SMFLDRN;
      <>I;
      );
      A(;
      L "idbEMX4".f[#p.child.EMX_SMFLDRN].p.read.mc.STATE;
      L "dbCONST".BLK.STATE.COMPLETED;
      <>I;
      );
      AN(;
      A(;
      L "dbCONST".BLK.CMD.START;
      L #childReqCMD.EMX_SMFLDRN;
      ==I;
      );
      A(;
      L "idbEMX4".f[#p.child.EMX_SMFLDRN].p.read.mc.STATE;
      L "idbEMX4".f[#p.child.EMX_SMFLDRN].p.write.mc.SUBS;
      ==I;
      );
      );
      );
      O(;
      A #selected_VESSEL_SY.S1;
      A "idbEMX2".f[#p.child.EMX_TRANSFER1].p.write.mc.ARMED;
      A "idbEMX2".f[#p.child.EMX_TRANSFER1].p.read.mc.FLOWPATH;
      A(;
      L "idbEMX2".f[#p.child.EMX_TRANSFER1].p.read.mc.STATE;
      L #childReqCMD.EMX_TRANSFER1;
      <>I;
      );
      A(;
      L "idbEMX2".f[#p.child.EMX_TRANSFER1].p.read.mc.STATE;
      L "dbCONST".BLK.STATE.COMPLETED;
      <>I;
      );
      AN(;
      A(;
      L "dbCONST".BLK.CMD.START;
      L #childReqCMD.EMX_TRANSFER1;
      ==I;
      );
      A(;
      L "idbEMX2".f[#p.child.EMX_TRANSFER1].p.read.mc.STATE;
      L "idbEMX2".f[#p.child.EMX_TRANSFER1].p.write.mc.SUBS;
      ==I;
      );
      );
      );
      O(;
      A #selected_VESSEL_SY.S2;
      A "idbEMX2".f[#p.child.EMX_TRANSFER2].p.write.mc.ARMED;
      A "idbEMX2".f[#p.child.EMX_TRANSFER2].p.read.mc.FLOWPATH;
      A(;
      L "idbEMX2".f[#p.child.EMX_TRANSFER2].p.read.mc.STATE;
      L #childReqCMD.EMX_TRANSFER2;
      <>I;
      );
      A(;
      L "idbEMX2".f[#p.child.EMX_TRANSFER2].p.read.mc.STATE;
      L "dbCONST".BLK.STATE.COMPLETED;
      <>I;
      );
      AN(;
      A(;
      L "dbCONST".BLK.CMD.START;
      L #childReqCMD.EMX_TRANSFER2;
      ==I;
      );
      A(;
      L "idbEMX2".f[#p.child.EMX_TRANSFER2].p.read.mc.STATE;
      L "idbEMX2".f[#p.child.EMX_TRANSFER2].p.write.mc.SUBS;
      ==I;
      );
      );
      );
      );
      JCN _noMismatch;

      S #flags.childMismatch;
      JC _noResetMismatch;

_noMismatch:      NOP 0;
      R #flags.childMismatch;
      R #p.read.mc.INTIL;

_noResetMismatch:      NOP 0;

NETWORK
TITLE = If child command changed, start timer to wait for child state
//------------------------------------------------------------------------//
// CHILD STATE TIMER   CHILD STATE TIMER   CHILD STATE TIMER   CHILD STAT //
//                                                                        //
// If any child command changed then start a timer to provide a grace     //
// period to allow the child device state to match the command (e.g. to   //
// allow a valve to move from closed to opened position).                 //
// Start the child state check timer if a command changed:                //
//------------------------------------------------------------------------//
      CALL #timeCheckChildState
      {time_type := 'Time'}
      (  IN                          := #flags.childMismatch ,
         PT                          := #p.read.bmc.transTime ,
         Q                           := #timeCheckChildStateExpired ,
         ET                          := #timeCheckChildStateElapsed
      );
      NOP 0;

NETWORK
TITLE = Block errors
//------------------------------------------------------------------------//
// Set the block start perimt error status if active:                     //
//------------------------------------------------------------------------//
      AN #p.read.bmc.permitStart;
      = #p.read.err.permitStart;

  //------------------------------------------------------------------------//
  // Set the child error status if active:                                  //
  //------------------------------------------------------------------------//
      A #flags.childInterlock;
      = #p.read.err.childInterlock;

  //------------------------------------------------------------------------//
  // Set the child unavailable error status if active:                      //
  //------------------------------------------------------------------------//
      A #flags.childUnavailable;
      = #p.read.err.childUnavailable;

  //------------------------------------------------------------------------//
  // Set the child state mismatch error status if active:                   //
  //------------------------------------------------------------------------//
      A #timeCheckChildStateExpired;
      = #p.read.err.childMismatch;
      JCN _noInternalIL;
      S #p.read.mc.INTIL;
_noInternalIL:      NOP 0;

  //------------------------------------------------------------------------//
  // Set the block error flag if anything gone wrong:                       //
  //------------------------------------------------------------------------//
      O #p.read.err.childInterlock;
      O #p.read.err.childMismatch;
      O #p.read.err.childSafeState;
      O #p.read.err.childUnavailable;
      O #p.read.err.permitStart;
      = #p.read.mc.ERROR;

NETWORK
TITLE = Pack the general block alarm bits
//------------------------------------------------------------------------//
// Pack the alarm bits into an integer for the HMI to read:               //
// Alarms are arranged in the following Little Endian order...            //
// Word   1                                0                              //
// Bit    0   1   2   3   4   5   6   7    8   9  10  11  12  13  14  15  //
// Order  9  10  11  12  13  14  15  16    1   2   3   4   5   6   7   8  //
//------------------------------------------------------------------------//
//    A #p.read.err.childInterlock;
//    = #b[8];
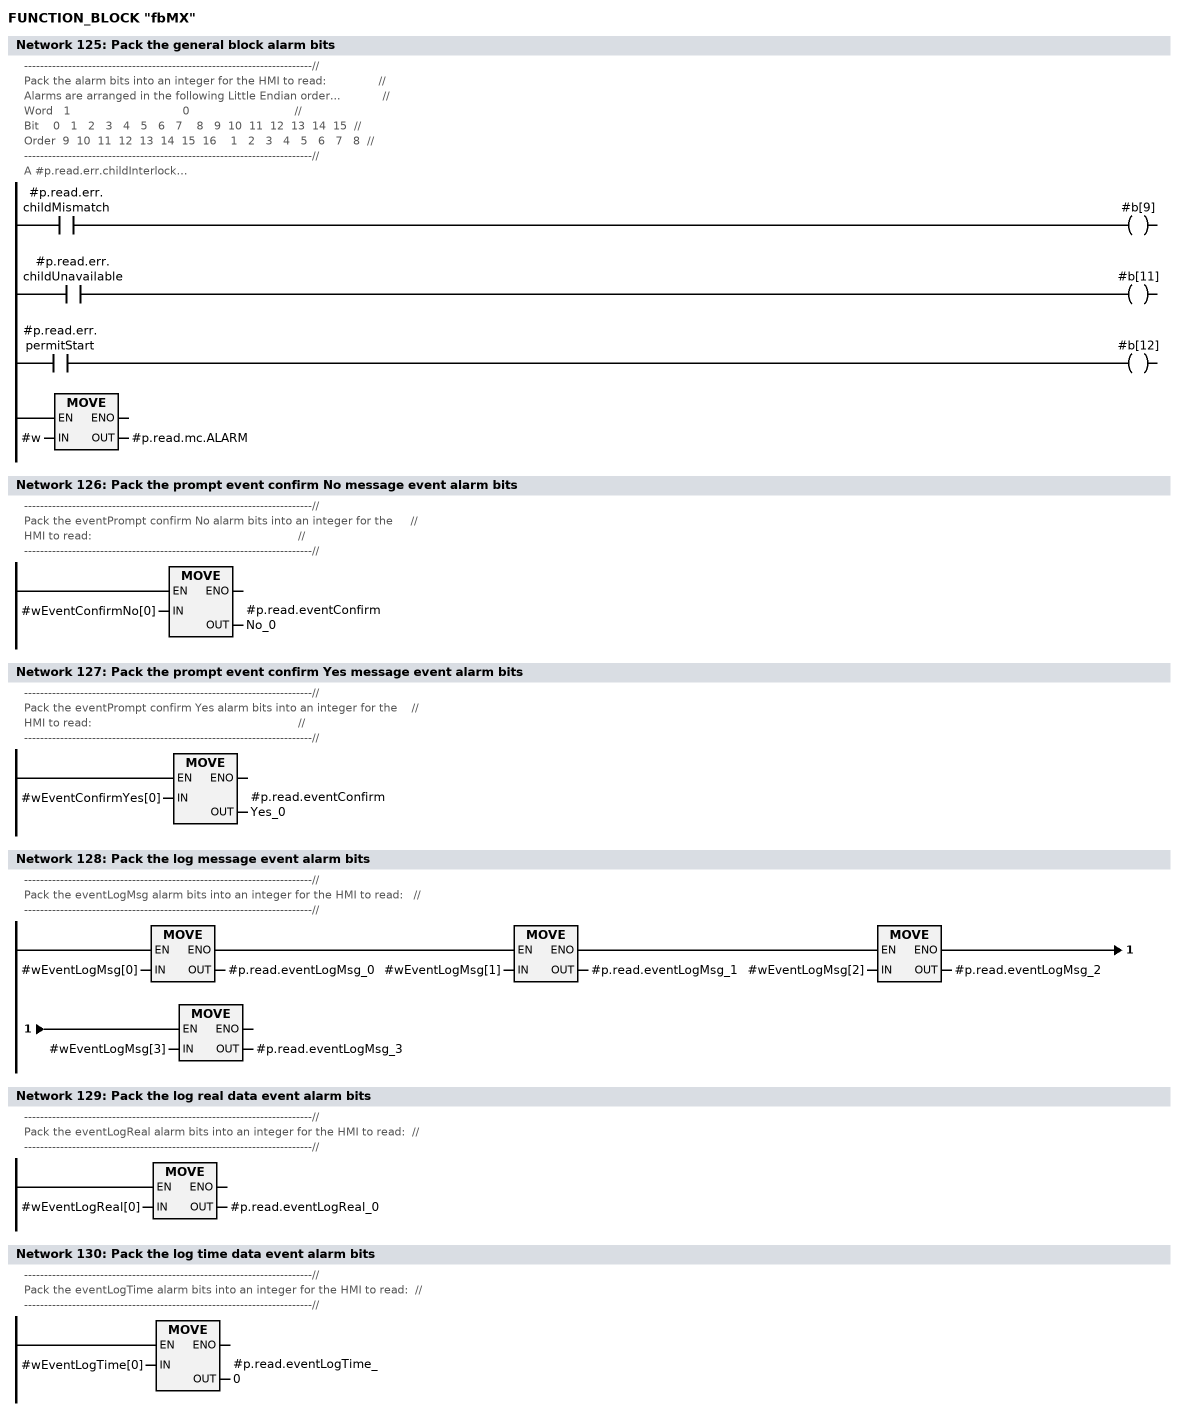
      A #p.read.err.childMismatch;
      = #b[9];
//    A #p.read.err.childSafeState;
//    = #b[10];
      A #p.read.err.childUnavailable;
      = #b[11];
      A #p.read.err.permitStart;
      = #b[12];
      L #w;
      T #p.read.mc.ALARM;

NETWORK
TITLE = Pack the prompt event confirm No message event alarm bits
//------------------------------------------------------------------------//
// Pack the eventPrompt confirm No alarm bits into an integer for the     //
// HMI to read:                                                           //
//------------------------------------------------------------------------//
      L #wEventConfirmNo[0];
      T #p.read.eventConfirmNo_0;

NETWORK
TITLE = Pack the prompt event confirm Yes message event alarm bits
//------------------------------------------------------------------------//
// Pack the eventPrompt confirm Yes alarm bits into an integer for the    //
// HMI to read:                                                           //
//------------------------------------------------------------------------//
      L #wEventConfirmYes[0];
      T #p.read.eventConfirmYes_0;

NETWORK
TITLE = Pack the log message event alarm bits
//------------------------------------------------------------------------//
// Pack the eventLogMsg alarm bits into an integer for the HMI to read:   //
//------------------------------------------------------------------------//
      L #wEventLogMsg[0];
      T #p.read.eventLogMsg_0;
      L #wEventLogMsg[1];
      T #p.read.eventLogMsg_1;
      L #wEventLogMsg[2];
      T #p.read.eventLogMsg_2;
      L #wEventLogMsg[3];
      T #p.read.eventLogMsg_3;

NETWORK
TITLE = Pack the log real data event alarm bits
//------------------------------------------------------------------------//
// Pack the eventLogReal alarm bits into an integer for the HMI to read:  //
//------------------------------------------------------------------------//
      L #wEventLogReal[0];
      T #p.read.eventLogReal_0;

NETWORK
TITLE = Pack the log time data event alarm bits
//------------------------------------------------------------------------//
// Pack the eventLogTime alarm bits into an integer for the HMI to read:  //
//------------------------------------------------------------------------//
      L #wEventLogTime[0];
      T #p.read.eventLogTime_0;

END_FUNCTION_BLOCK

